FUNCTION_BLOCK ProductPriceConverter (* Basic Function Block Type *)
  (* Standard: 61499-2 *)
  (* Version 0.3, 2009-09-15, JHC, Holobloc Inc, Changed transition priorities. *)
  (* Version 0.2, 2003-12-04, JHC, Rockwell Automation, Renamed for better indexing. *)
  (* Version 0.1, 2002-11-05, JHC, Rockwell Automation, Corrected missing ST element in Algorithm REQ. *)
  (* Version 0.0, 2000-05-30, JHC, Rockwell Automation *)
  (* Compiler header: package fb.rt.template; *)
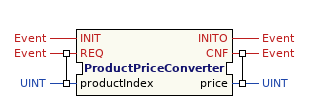
  EVENT_INPUT
    INIT; (* Initialization Request *)
    REQ WITH productIndex; (* Normal Execution Request *)
  END_EVENT
  EVENT_OUTPUT
    INITO; (* Initialization Confirm *)
    CNF WITH price; (* Execution Confirmation *)
  END_EVENT
  VAR_INPUT
    productIndex : UINT;
  END_VAR
  VAR_OUTPUT
    price : UINT;
  END_VAR
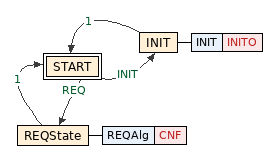
  EC_STATES
    START; (* Initial State *)
    INIT : INIT -> INITO; (* Initialization *)
    REQState : REQAlg -> CNF; (* Normal execution *)
  END_STATES
  EC_TRANSITIONS
    INIT TO START := 1;
    START TO REQState := REQ;
    START TO INIT := INIT;
    REQState TO START := 1;
  END_TRANSITIONS
  ALGORITHM INIT IN ST: (* Initialization algorithm *)

  END_ALGORITHM
  ALGORITHM REQAlg IN ST: (* Normally executed algorithm *)
CASE productIndex OF
3:
	price:=10;
1:
	price:=20;
2:
	price:=30;
ELSE
	price:=1;
END_CASE;
  END_ALGORITHM
END_FUNCTION_BLOCK
